(* IEC 61131-3 sources: AXOpen/src/data/tests/AXOpen.Data.Tests_L1/ax/src, 2 files *)

(* ---- configuration.st ---- *)
USING AXOpen.Data;
CONFIGURATION MyConfiguration
    TASK Main(Interval := T#10ms, Priority := 1);
    PROGRAM P1 WITH Main: MyProgram;

    VAR_GLOBAL

        {S7.extern=ReadWrite}
        DataExchange : Tests_L1.DataExchange.DataExchangeContext;

        {S7.extern=ReadWrite}
        Fragments : Tests_L1.FragmentData.FragmentDataContext;

        {S7.extern=ReadWrite}
        Distributed : Tests_L1.Distributed.DistributedDataContext;

        {S7.extern=ReadWrite}
        Persistent : Tests_L1.PersistentData.PersistentDataContext;

    END_VAR
END_CONFIGURATION

(* ---- program.st ---- *)
PROGRAM MyProgram
    VAR_EXTERNAL
        DataExchange : Tests_L1.DataExchange.DataExchangeContext;
        Fragments : Tests_L1.FragmentData.FragmentDataContext;
        Distributed : Tests_L1.Distributed.DistributedDataContext;
        Persistent : Tests_L1.PersistentData.PersistentDataContext;

    END_VAR

    DataExchange.Run();
    Fragments.Run();
    Distributed.Run();
    Persistent.Run();

END_PROGRAM
